(* CoDeSys 2.3.9.47 project: wtp_new.pro *)
(* Libraries: STANDARD.LIB 5.6.98 12:03:02 *)

(* Task configuration *)
TASK Standard (PRIORITY := 0, INTERVAL := T#10ms);
	MAIN
END_TASK

(* POU MAIN, ST *)
PROGRAM MAIN
VAR
	InletEqPump1 : EQ_PUMP;
	InletMixer1 : IN_MIXER;

	Screening : INLET_SCREENING;
END_VAR
InletEqPump1();
InletMixer1();
Screening();
GRIT_REMOVAL();
END_PROGRAM

(* POU EQ_PUMP, ST *)
FUNCTION_BLOCK EQ_PUMP
VAR_INPUT
END_VAR
VAR_OUTPUT
END_VAR
VAR
	EQFloatSensorLO: BOOL;
	EQFloatSensorOP: BOOL;
	EQFLoatSensorHI: BOOL;
	SLSensorOverflow: BOOL;
	EQPumpDuty: BOOL;
	SBRFloatSensorHi: BOOL;
	EQPumpStandby: BOOL;
	EQFLoatSensorDry: BOOL;

	CriticalAlarm_EQFloatSensorHi: BOOL;
	WarningAlarm_EQFloatSensorDry: BOOL;
	CriticalAlarm_EQFloatSensorDry: BOOL;
	WarningAlarm_EQFloatSensorLow: BOOL;

	Pump : DutyStandby;
	Reset:BOOL;
END_VAR
IF EQFloatSensorLO THEN
	IF EQFloatSensorOP THEN
		EQPumpDuty := TRUE;
		IF EQFloatSensorHi THEN
			IF SBRFloatSensorHi OR SLSensorOverflow THEN
				EQPumpDuty := FALSE;
				EQPumpStandby := FALSE;
			END_IF
			CriticalAlarm_EQFloatSensorHi := TRUE;
		END_IF
	ELSE
		EQPumpDuty := FALSE;
		EQPumpStandby := FALSE;
	END_IF
ELSE
	EQPumpDuty := FALSE;
	EQPumpStandby := FALSE;
	IF EQFLoatSensorDry THEN
		WarningAlarm_EQFloatSensorLow :=TRUE;
	ELSE
		CriticalAlarm_EQFloatSensorDry := TRUE;
	END_IF
END_IF

Pump(
	Duty:=EQPumpDuty ,
	Standby:=EQPumpStandby );


IF Reset THEN
	CriticalAlarm_EQFloatSensorHi:=FALSE;
	WarningAlarm_EQFloatSensorDry:=FALSE;
	CriticalAlarm_EQFloatSensorDry:=FALSE;
	WarningAlarm_EQFloatSensorLow:=FALSE;
END_IF
END_FUNCTION_BLOCK

(* POU PARTS/DutyStandby, ST *)
FUNCTION_BLOCK DutyStandby
VAR_INPUT
END_VAR
VAR_OUTPUT
END_VAR
VAR
	timer: TON;
	timer2: TON;

	Warning_DutyNotStart: BOOL;

	DutyCmd: BOOL;
	DutyRemote: BOOL;
	DutyOverload: BOOL;
	DutyIncomplete: BOOL;
	DutyStat: BOOL;
	StandbyCmd: BOOL;
	StandbyRemote: BOOL;
	StandbyOverload: BOOL;
	StandbyIncomplete: BOOL;
	StandbyStat: BOOL;

	Warning_StandbyNotStart: BOOL;
	CriticalAlarm_StartingFailed: BOOL;
	Critical_DutyNotStop: BOOL;
	Critical_StandbyNotStop: BOOL;

	ESTOP : BOOL;
	Reset: BOOL;
END_VAR
VAR_IN_OUT

	Duty: BOOL;
	Standby: BOOL;
END_VAR
IF Duty THEN
	IF DutyRemote THEN
		DutyCmd := TRUE;
		timer(IN:=TRUE , PT:=T#2s);
		IF timer.Q THEN
			IF DutyOverload OR DutyIncomplete OR NOT DutyStat THEN
				Warning_DutyNotStart := TRUE;
				Standby := TRUE;
			ELSE
				Standby := FALSE;
			END_IF
			timer(IN:=FALSE);
		END_IF
	END_IF
ELSE
	IF DutyRemote THEN
		DutyCmd := FALSE;
		timer(IN:=TRUE , PT:=T#2s);
			IF timer.Q THEN
			timer(IN:=FALSE , PT:=T#2s);
				IF DutyStat THEN
					Critical_DutyNotStop := TRUE;
					ESTOP := TRUE;
				END_IF
			END_IF
	END_IF
END_IF

IF Standby THEN
	IF StandbyRemote THEN
		StandbyCmd := TRUE;
		timer2(IN:=TRUE , PT:=T#2s);
		IF timer.Q THEN
			timer2(IN:=FALSE);
			IF StandbyOverload OR StandbyIncomplete OR NOT StandbyStat THEN
				Warning_StandbyNotStart := TRUE;
				IF DutyOverload OR DutyIncomplete THEN
					CriticalAlarm_StartingFailed :=TRUE;
				END_IF
			END_IF
		END_IF
	END_IF
ELSE
	IF StandbyRemote THEN
		StandbyCmd := FALSE;
		timer2(IN:=TRUE , PT:=T#2s);
			IF timer2.Q THEN
			timer2(IN:=FALSE , PT:=T#2s);
				IF StandbyStat THEN
					Critical_StandbyNotStop := TRUE;
					ESTOP := TRUE;
				END_IF
			END_IF
	END_IF
END_IF

IF reset THEN
Warning_DutyNotStart:= FALSE;
Warning_StandbyNotStart:= FALSE;
CriticalAlarm_StartingFailed:= FALSE;
Critical_DutyNotStop:= FALSE;
ESTOP:= FALSE;
Critical_StandbyNotStop:= FALSE;
END_IF
END_FUNCTION_BLOCK

(* POU IN_MIXER, ST *)
FUNCTION_BLOCK IN_MIXER
VAR_INPUT
END_VAR
VAR_OUTPUT
END_VAR
VAR
	Mixer : DutyStandby;
	MixerFloatSensorLO: BOOL;
	MixerFloatSensorHi: BOOL;
	EQMixerDuty: BOOL;
	EQMixerStandby: BOOL;
END_VAR
IF MixerFloatSensorLO THEN
	IF MixerFloatSensorHi THEN
		EQMixerDuty := TRUE;
	ELSE
		EQMixerDuty := FALSE;
		EQMixerStandby := FALSE;
	END_IF
ELSE
		EQMixerDuty := FALSE;
		EQMixerStandby := FALSE;
END_IF
Mixer(
	Duty:=EQMixerDuty ,
	Standby:=EQMixerStandby );
END_FUNCTION_BLOCK

(* POU INLET_SCREENING, ST *)
FUNCTION_BLOCK INLET_SCREENING
VAR_INPUT
END_VAR
VAR_OUTPUT
END_VAR
VAR
	fbPenstock : Penstock;
	PenstockDuty: BOOL;
	PenstockStandby: BOOL;
	Reset: BOOL;

	fbFineScreen : DutyStandbyFineScreen;
	FineScreenDuty: BOOL;
	FineScreenStandby: BOOL;
	WaterSprayScreenDuty: BOOL;
	WaterSprayScreenStandby: BOOL;
	ScrewConveyor: BOOL;
	ScrewCompactor: BOOL;

	fbWaterSprayScreenDuty : WaterSprayScreen;
	fbWaterSprayScreenStandby:WaterSprayScreen;

	fbContinuousWaterSpray : ContinuousWaterSpray;

	ContWaterSpray: BOOL := TRUE;

END_VAR
fbPenstock(
	Duty:= PenstockDuty,
	Standby:= PenstockStandby);

fbFineScreen(
	Duty:=FineScreenDuty ,
	Standby:=FineScreenStandby ,
	WaterSprayScreenDuty:= WaterSprayScreenDuty,
	WaterSprayScreenStandby:=WaterSprayScreenStandby ,
	PenstockStandby:= PenstockDuty,
	PenstockDuty:=PenstockStandby ,
	ScrewConveyor:=ScrewConveyor ,
	ScreenCompactor:=ScrewCompactor );

fbWaterSprayScreenDuty(WaterSprayScreen:= WaterSprayScreenDuty);
fbWaterSprayScreenStandby(WaterSprayScreen:=WaterSprayScreenStandby );

fbContinuousWaterSpray(ContWS:=ContWaterSpray );
END_FUNCTION_BLOCK

(* POU PARTS/Penstock, ST *)
FUNCTION_BLOCK Penstock
VAR_INPUT
END_VAR
VAR_OUTPUT
END_VAR
VAR
	timer1:TON;

	DutyCommand: BOOL;
	DutyStat: BOOL;
	Warning_DutyNotStart: BOOL;
	Warning_DutyNotStop: BOOL;

	StandbyCommand: BOOL;
	timer2: TON;
	StandbyStat: BOOL;
	Warning_StandbyNotStart: BOOL;
	Warning_StandbyNotStop: BOOL;
	Reset:BOOL;
END_VAR
VAR_IN_OUT
	Duty: BOOL;
	Standby: BOOL;

END_VAR
IF Duty THEN
	DutyCommand := TRUE;
	timer1(IN:=TRUE,PT:=T#2s);
		IF timer1.Q THEN
		timer1(IN:=FALSE,PT:=T#2s);
			IF  NOT DutyStat  THEN
				Warning_DutyNotStart:=TRUE;
			END_IF
		END_IF
ELSE
	DutyCommand := FALSE;
	timer1(IN:=TRUE,PT:=T#2s);
		IF timer1.Q THEN
		timer1(IN:=FALSE,PT:=T#2s);
			IF  DutyStat  THEN
				Warning_StandbyNotStart:=TRUE;
			END_IF
		END_IF
END_IF

IF Standby THEN
	StandbyCommand := TRUE;
	timer2(IN:=TRUE,PT:=T#2s);
		IF timer2.Q THEN
		timer2(IN:=FALSE,PT:=T#2s);
			IF  NOT StandbyStat  THEN
				Warning_StandbyNotStart:=TRUE;
			END_IF
		END_IF
ELSE
	StandbyCommand := FALSE;
	timer2(IN:=TRUE,PT:=T#2s);
		IF timer1.Q THEN
		timer2(IN:=FALSE,PT:=T#2s);
			IF  StandbyStat  THEN
				Warning_StandbyNotStop:=TRUE;
			END_IF
		END_IF
END_IF

IF reset THEN
Warning_DutyNotStart:=FALSE;
Warning_DutyNotStop:=FALSE;
Warning_StandbyNotStart:=FALSE;
Warning_StandbyNotStop:=FALSE;
END_IF
END_FUNCTION_BLOCK

(* POU PARTS/DutyStandbyFineScreen, ST *)
FUNCTION_BLOCK DutyStandbyFineScreen
VAR_INPUT
END_VAR
VAR_OUTPUT
END_VAR
VAR
	timer: TON;
	timer2: TON;

	Warning_DutyNotStart: BOOL;

	DutyCmd: BOOL;
	DutyRemote: BOOL;
	DutyOverload: BOOL;
	DutyIncomplete: BOOL;
	DutyStat: BOOL;
	StandbyCmd: BOOL;
	StandbyRemote: BOOL;
	StandbyOverload: BOOL;
	StandbyIncomplete: BOOL;
	StandbyStat: BOOL;

	Warning_StandbyNotStart: BOOL;
	CriticalAlarm_StartingFailed: BOOL;
	Critical_DutyNotStop: BOOL;
	Critical_StandbyNotStop: BOOL;

	ESTOP : BOOL;

	timer11: TON;
	timer22: TON;
	timer3: TON;
	Reset: BOOL;
END_VAR
VAR_IN_OUT

	Duty: BOOL;
	Standby: BOOL;

	WaterSprayScreenDuty: BOOL;
	WaterSprayScreenStandby: BOOL;
	PenstockStandby: BOOL;
	PenstockDuty: BOOL;
	ScrewConveyor: BOOL;
	ScreenCompactor: BOOL;
END_VAR
IF Duty THEN
	IF DutyRemote THEN
		DutyCmd := TRUE;
		timer(IN:=TRUE , PT:=T#2s);
		IF timer.Q THEN
			IF DutyOverload OR DutyIncomplete OR NOT DutyStat THEN
				Warning_DutyNotStart := TRUE;
				Standby := TRUE;
			ELSE
				Standby := FALSE;
				WaterSprayScreenDuty := TRUE;
				PenstockDuty := TRUE;
				PenstockStandby := FALSE;
			END_IF
			timer(IN:=FALSE);
		END_IF
	END_IF
ELSE
	IF DutyRemote THEN
		timer(IN:=TRUE , PT:=T#2m);
		IF timer.Q THEN
			DutyCmd := FALSE;
			WaterSprayScreenDuty := FALSE;
			timer11(IN:=TRUE , PT:=T#2s);
			IF timer11.Q THEN
				timer(IN:=FALSE);
				timer11(IN:=FALSE);
					IF DutyStat THEN
						Critical_DutyNotStop := TRUE;
						ESTOP := TRUE;
					END_IF
			END_IF
		END_IF
	END_IF
END_IF

IF Standby THEN
	IF StandbyRemote THEN
		StandbyCmd := TRUE;
		timer2(IN:=TRUE , PT:=T#2s);
		IF timer.Q THEN
			timer2(IN:=FALSE);
			IF StandbyOverload OR StandbyIncomplete OR NOT StandbyStat THEN
				Warning_StandbyNotStart := TRUE;
				IF DutyOverload OR DutyIncomplete THEN
					CriticalAlarm_StartingFailed :=TRUE;
					ScrewConveyor:=FALSE;
				ELSE
					Duty := TRUE;
				END_IF
			ELSE
				WaterSprayScreenStandby := TRUE;
				PenstockDuty := FALSE;
				PenstockStandby:=TRUE;
				Duty:= FALSE;
			END_IF
		END_IF
	END_IF
ELSE
	IF StandbyRemote THEN
		timer2(IN:=TRUE , PT:=T#2m);
		IF timer2.Q THEN
			StandbyCmd := FALSE;
			timer22(IN:=TRUE , PT:=T#2s);
				IF timer22.Q THEN
					timer2(IN:=FALSE);
					timer22(IN:=FALSE);
						IF StandbyStat THEN
							Critical_StandbyNotStop := TRUE;
							ESTOP := TRUE;
						END_IF
				END_IF
		END_IF
	END_IF
END_IF

IF NOT duty AND NOT standby THEN
	timer3(IN:=TRUE,pt:=T#5m);
	IF timer3.Q THEN
		ScrewConveyor:=FALSE;
		ScreenCompactor:=FALSE;
	END_IF
END_IF


IF reset THEN
Warning_DutyNotStart:= FALSE;
Warning_StandbyNotStart:= FALSE;
CriticalAlarm_StartingFailed:= FALSE;
Critical_DutyNotStop:= FALSE;
ESTOP:= FALSE;
Critical_StandbyNotStop:= FALSE;
END_IF
END_FUNCTION_BLOCK

(* POU PARTS/WaterSprayScreen, ST *)
FUNCTION_BLOCK WaterSprayScreen
VAR_INPUT
END_VAR
VAR_OUTPUT
END_VAR
VAR


	timer1: TON;
	timer2: TON;
	timer3: TON;
	timer4:TON;
	CriticalAlarm_NotClose: BOOL;
	WarningAlarm_NotOpen: BOOL;

	Warning_NotClose: BOOL;
	WaterSprayScreenCmdi: BOOL;

	WaterSprayScreenCmd: BOOL;
	WaterSprayScreenClose: BOOL;
	WaterSprayScreenOpen: BOOL;
	Reset: BOOL;
END_VAR
VAR_IN_OUT
	WaterSprayScreen:BOOL;
END_VAR
IF WaterSprayScreen THEN
	WaterSprayScreenCmdi := TRUE;
	timer1(IN:=TRUE,PT:=T#2s);
	IF  timer1.Q THEN
		IF WaterSprayScreenOpen THEN
			timer2(IN:=TRUE,PT:=T#1m);
			IF timer2.Q THEN
				WaterSprayScreenCmdi := FALSE;
				timer3(IN:=TRUE,PT:=T#5m);
				IF timer3.Q THEN
					timer1(IN:=FALSE);
					timer2(IN:=FALSE);
					timer3(IN:=FALSE);
				END_IF
			END_IF
		ELSE
			WarningAlarm_NotOpen := TRUE;
			timer1(IN:=FALSE,PT:=T#2s);
		END_IF
	END_IF
ELSE
	WaterSprayScreenCmdi := FALSE;
	timer1(IN:=FALSE);
	timer2(IN:=FALSE);
	timer3(IN:=FALSE);
END_IF

IF WaterSprayScreenCmdi THEN
	WaterSprayScreenCmd := TRUE;
ELSE
	WaterSprayScreenCmd := FALSE;
	timer4(in:=TRUE,PT:=T#2s);
		IF timer4.Q THEN
		timer4(in:=FALSE,PT:=T#2s);
			IF NOT WaterSprayScreenClose THEN
				IF WaterSprayScreenOpen THEN
					CriticalAlarm_NotClose := TRUE;
				ELSE
					Warning_NotClose := TRUE;
				END_IF
			END_IF
		END_IF
END_IF

IF Reset THEN
	CriticalAlarm_NotClose:=FALSE;
	WarningAlarm_NotOpen:=FALSE;
	Warning_NotClose:=FALSE;
END_IF
END_FUNCTION_BLOCK

(* POU PARTS/ContinuousWaterSpray, ST *)
FUNCTION_BLOCK ContinuousWaterSpray
VAR_INPUT
END_VAR
VAR_OUTPUT
END_VAR
VAR
	ContWSCmd: BOOL;

	ContWSOpen: BOOL;
	ContWSClose: BOOL;

	Warning_NotStart: BOOL;
	Critical_NotClose: BOOL;
	Warning_NotClose: BOOL;

	timer1: TON;
	Reset: BOOL;
END_VAR
VAR_IN_OUT
	ContWS: BOOL;
END_VAR
IF ContWS THEN
	ContWSCmd := TRUE;
	timer1(in:=TRUE,pt:=t#2s);
	IF timer1.Q THEN
		timer1(in:=FALSE);
		IF NOT ContWSOpen THEN
			Warning_NotStart := TRUE;
		END_IF
	END_IF
ELSE
	ContWSCmd := FALSE;
	timer1(in:=TRUE,pt:=t#2s);
	IF timer1.Q THEN
		timer1(in:=FALSE);
		IF NOT ContWSClose THEN
			IF ContWSOpen THEN
				Critical_NotClose  := TRUE;
			ELSE
				Warning_NotClose := TRUE;
			END_IF
		END_IF
	END_IF
END_IF

IF Reset THEN
	Warning_NotStart:=FALSE;
	Critical_NotClose:=FALSE;
	Warning_NotClose:=FALSE;
END_IF
END_FUNCTION_BLOCK

(* POU GRIT_REMOVAL, ST *)
PROGRAM GRIT_REMOVAL
VAR
	bStreamlineHi: BOOL;
	bStreamlineSensorHiA: BOOL;
	bStreamlineSensorHiB: BOOL;
	bSuctionValve: BOOL;
	bAirBlower: BOOL;
	bClassifier: BOOL;
	TStreamlineHi: TOF;

	fbAirBlower: AirBlower;
END_VAR
bStreamlineHi := bStreamlineSensorHiA OR bStreamlineSensorHiB;
bSuctionValve := bStreamlineHi;
bAirBlower := bStreamlineHi;
bClassifier := TStreamlineHi.Q;
TStreamlineHi(IN:=bStreamlineHi , PT:=T#5m );
fbAirBlower(IN:=bAirBlower );
END_PROGRAM

(* POU PARTS/AirBlower, ST *)
FUNCTION_BLOCK AirBlower
VAR_INPUT
	IN : BOOL;
END_VAR
VAR_OUTPUT
END_VAR
VAR

	DutyOverload: BOOL;
	DutyIncomplete: BOOL;
	StandbyOverload: BOOL;
	StandbyIncomplete: BOOL;
	DutyStarted: BOOL;
	StandbyStarted: BOOL;


	TCheckDutyON: TON;
	TCheckStandbyON: TON;
	dutyTimer: TON;
	standbyTimer: TON;

	startDuty: BOOL;
	startStandby: BOOL;

	WarningDuty: BOOL;
	WarningStandby: BOOL;
	CriticalAlarmStart: BOOL;
	StopTimer: TON;
	CriticalAlarmStop: BOOL;
	checkDuty: BOOL;
	checkStandby: BOOL;
END_VAR
startDuty := IN AND NOT startStandby ;
dutyTimer(IN := startDuty AND NOT dutyTimer.Q , PT:=T#2s);
TCheckDutyON(IN := startDuty AND NOT TCheckDutyON.Q , PT:=T#60m);
checkDuty := dutyTimer.Q OR TCheckDutyON.Q;
WarningDuty := SEL(checkDuty,WarningDuty, (DutyOverload OR DutyIncomplete) OR NOT(DutyStarted));
startDuty := SEL( checkDuty,  startDuty,   NOT (WarningDuty OR TCheckDutyON.Q) ) ;


startStandby := (IN AND NOT startDuty) AND NOT(startDuty AND startStandby);
standbyTimer(IN := startStandby AND NOT standbyTimer.Q, PT:=T#2s);
TCheckStandbyON(IN := startStandby AND NOT TCheckStandbyON.Q , PT:=T#60m);
checkStandby := standbyTimer.Q OR TCheckStandbyON.Q;
WarningStandby := SEL(checkStandby, WarningStandby, (StandbyOverload OR StandbyIncomplete) OR NOT(StandbyStarted));
startStandby := SEL(checkStandby,startStandby ,NOT (WarningStandby OR TCheckStandbyON.Q)) ;


CriticalAlarmStart := IN AND SEL(checkDuty OR checkStandby,CriticalAlarmStart, WarningStandby AND WarningDuty);
StopTimer(IN := NOT IN AND NOT StopTimer.Q , PT:=T#2s);
CriticalAlarmStop := NOT IN AND SEL(StopTimer.Q,CriticalAlarmStop,(DutyStarted OR StandbyStarted));
END_FUNCTION_BLOCK

(* POU PARTS/GritRemovalSuctionValve, ST *)
FUNCTION_BLOCK GritRemovalSuctionValve
VAR_INPUT
	ON: BOOL;
	WarningDutyB: BOOL;
END_VAR
VAR_OUTPUT
END_VAR
VAR
	AirBlowerDuty: BOOL;
	Standby: BOOL;
	Start: BOOL;

	SuctionValveDutyA: BOOL;
	PenstockDutyA: BOOL;
	SuctionValveStandbyA: BOOL;
	PenstockStandbyA: BOOL;
	SuctionValveDutyB: BOOL;
	PenstockDutyB: BOOL;
	SuctionValveStandbyB: BOOL;
	PenstockStandbyB: BOOL;
	Timer1: TON;
	Timer2: TON;
	Timer3: TON;
	Timer4: TON;
	Timer1f: TON;
	Timer2f: TON;
	Timer3f: TON;
	Timer4f: TON;
	WarningDutyA: BOOL;
	SuctionValveDutyAStat: BOOL;
	WarningStandbyA: BOOL;
	SuctionValveStandbyAStat: BOOL;
	WarningStandbyB: BOOL;
	SuctionValveDutyBStat: BOOL;
	SuctionValveStandbyBStat: BOOL;
	bAirBlower: BOOL;
	AirBlowerStandby: BOOL;
	WarningDutyStopA: BOOL;
	WarningStandbyStopA: BOOL;
	WarningDutyStopB: BOOL;
	WarningStandbyStopB: BOOL;
END_VAR
bAirBlower := AirBlowerDuty OR AirBlowerStandby;
Start := bAirBlower AND ON;

SuctionValveDutyA := start AND PenstockDutyA;
SuctionValveStandbyA := start AND PenstockStandbyA;
SuctionValveDutyB := start AND PenstockDutyB;
SuctionValveStandbyB := start AND PenstockStandbyB;

Timer1(IN:=SuctionValveDutyA , PT:=T#2s);
WarningDutyA := Timer1.Q AND NOT SuctionValveDutyAStat;
Timer2(IN:=SuctionValveStandbyA , PT:=T#2s);
WarningStandbyA := Timer2.Q AND NOT SuctionValveStandbyAStat;
Timer3(IN:=SuctionValveDutyA , PT:=T#2s);
WarningDutyB := Timer3.Q AND NOT SuctionValveDutyBStat;
Timer4(IN:=SuctionValveStandbyA , PT:=T#2s);
WarningStandbyB := Timer4.Q AND NOT SuctionValveStandbyBStat;


Timer1f(IN:=NOT SuctionValveDutyA , PT:=T#2s);
WarningDutyStopA := Timer1f.Q AND SuctionValveDutyAStat;
Timer2f(IN:=NOT SuctionValveStandbyA , PT:=T#2s);
WarningStandbyStopA := Timer2f.Q AND SuctionValveStandbyAStat;
Timer3f(IN:=NOT SuctionValveDutyA , PT:=T#2s);
WarningDutyStopB := Timer3f.Q AND SuctionValveDutyBStat;
Timer4f(IN:=NOT SuctionValveStandbyA , PT:=T#2s);
WarningStandbyStopB := Timer4f.Q AND SuctionValveStandbyBStat;
END_FUNCTION_BLOCK
